{attribute 'GeneratedUsingTerminal: EL3356-0030-0025'}
{attribute addProperty BoxType "EL3356-0030-0025"}
{attribute addProperty Id "StatusAT %I*Status_7BCDA9217"}
{attribute addProperty CRC "3235971242"}
{attribute addProperty Size "7"}
TYPE RMB_Status_C0E100AA :
STRUCT
	{attribute addProperty Name "Status"}
	Status AT %I* : Status_7BCDA921;
END_STRUCT
END_TYPE

(* stored: Version 1.2.0.0, ProductVersion 3.1.4024.9
   DUT RMB_Status_C0E100AA: Id {e8b84986-10a7-4925-b30a-f8b9af4cd790} *)
